TYPE MyStruct :
STRUCT
	MyBit : BIT;
END_STRUCT
END_TYPE

(* stored: Version 1.1.0.1, ProductVersion 3.1.4024.12
   DUT MyStruct: Id {a5721eb2-c8a8-4178-a856-ee49aec60912} *)
